FUNCTION_BLOCK OpcTagWritingHandler
VAR_INPUT
END_VAR
VAR_OUTPUT
END_VAR
VAR
	serialCommReadData : ST_SerialCommReadData;
	onOffValveValues : ST_ExtractiveOnOffValveValues;
END_VAR


// Reactor temperature
GVL_OPC.OPC_ReactorTemperature := GVL_IO.reactorTemperatureUpper;
GVL_OPC.OPC_TemperatureContactor := GVL_IO.reactorTemperatureContactor;
IF ReactorTemperatureController._autoControlSelected THEN
	GVL_OPC.OPC_ReactorTemperatureSetpoint := REAL_TO_INT(ReactorTemperatureController._temperatureSetpoint);
ELSE
	GVL_OPC.OPC_ReactorTemperatureSetpoint := 0;
END_IF

// Reactor pressure
GVL_OPC.OPC_ReactorPressure := ReactorLevelAndPressureController.iPressureScaledValue;

// Valves
GVL_OPC.OPC_SlurryInletValve := GVL_IO.reactorInletValve;
GVL_OPC.OPC_SlurryOutletValve := GVL_IO.reactorOutletValve;
onOffValveValues := ReactorLevelAndPressureController.ExtractiveOnOffValveValues;
GVL_OPC.OPC_ExtractiveOutletOnOffValve := onOffValveValues.open;
GVL_OPC.OPC_ExtractiveControlValveOpening := TO_INT(ReactorLevelAndPressureController.ControlValveOpening);

// Serial comm data
serialCommReadData := SerialCommunicationController.serialCommReadData;
GVL_OPC.OPC_CO2VolumetricFlow := serialCommReadData.flowMeasurement;
GVL_OPC.OPC_PumpingPressure := serialCommReadData.pumpingPressureMeasurement;
GVL_OPC.OPC_PumpingPressureSetpoint := serialCommReadData.pumpingPressureSetpoint;
GVL_OPC.OPC_PreHeaterTemperature := serialCommReadData.preHeaterTemperatureMeasurement;
GVL_OPC.OPC_PreHeaterTemperatureSetpoint := serialCommReadData.preHeaterTemperatureSetpoint;
GVL_OPC.OPC_SeparatorTemperature := serialCommReadData.separatorTemperatureMeasurement;
GVL_OPC.OPC_SeparatorTemperatureSetpoint := serialCommReadData.separatorTemperatureSetpoint;

END_FUNCTION_BLOCK

(* stored: Version 1.1.0.1, ProductVersion 3.1.4024.9
   POU OpcTagWritingHandler: Id {016e686a-2418-421a-bdfe-907d5d5f760a}, SpecialFunc None *)
